{attribute 'pack_mode' := '1'}
TYPE DUT_EpicsValueDouble :
STRUCT
	stMetadata : DUT_EpicsValueMetadata;
	fValue : LREAL;
END_STRUCT
END_TYPE

(* stored: Version 1.1.0.1, ProductVersion 3.1.4022.18
   DUT DUT_EpicsValueDouble: Id {0a11fb73-3372-4e4c-98d0-e393f1d5d024} *)
